// ---- MODULE/ACTOR_VALVE/PNEUMATIC_ACTOR/VISU/VisuCylinderHorLeft.TcVIS
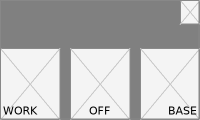
VISUALIZATION VisuCylinderHorLeft  // 200x120
VAR_IN_OUT
	fbVisuCylinder: FB_VISU_CYLINDER;
END_VAR
    Textfield (0,15 200x20), "%s", text variable: fbVisuCylinder.strInfo, colour toggle: fbVisuCylinder.stEvent.bEventActive
    Textfield (0,0 200x14), "%s", text variable: fbVisuCylinder.strFullObjName
    Image (143,85 52x30), invisible if: fbVisuCylinder.bBaseArrowInvisible, image: VisuSymbols.Symbols.ArrowBoldRight
        p2175578022: fbVisuCylinder.dwFrameColorBase
    Image (85,85 52x30), invisible if: fbVisuCylinder.bWorkArrowInvisible, image: VisuSymbols.Symbols.ArrowBoldLeft
        p2175578022: fbVisuCylinder.dwFrameColorWork
    Group (90,35 105x40)
        p3560616238: fbVisuCylinder.iMove
        RoundedRectangle (-10,10 100x20)
        RoundedRectangle (80,0 20x40)
    Rectangle (85,35 105x40)
        OnMouseClick: execute { fbVisuCylinder.bFrameInvisible:=false; }
    Frame (0,0 200x120), invisible if: fbVisuCylinder.bFrameInvisible, frame switch variable: fbVisuCylinder.iFrame
        shows VisuCylinderHorLeftCtrl(fbVisuCylinder := fbVisuCylinder)
END_VISUALIZATION

// ---- MODULE/ACTOR_VALVE/PNEUMATIC_ACTOR/VISU/VisuCylinderHorLeftCtrl.TcVIS
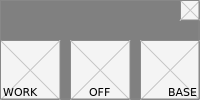
VISUALIZATION VisuCylinderHorLeftCtrl  // 200x100
VAR_IN_OUT
	fbVisuCylinder: FB_VISU_CYLINDER;
END_VAR
    Rectangle (0,0 200x100)
    Image (140,40 60x60), "BASE", image: VisuSymbols.Symbols.TriangleRight
        OnMouseClick: execute {
            fbVisuCylinder.bMoveToBase:=TRUE;
            fbVisuCylinder.bMoveToWork:=FALSE;
            fbVisuCylinder.bAllOff:=false;
            fbVisuCylinder.bFrameInvisible:= true;
        }
    Image (0,40 60x60), "WORK", image: VisuSymbols.Symbols.TriangleLeft
        OnMouseClick: execute {
            fbVisuCylinder.bMoveToWork:=TRUE;
            fbVisuCylinder.bMoveToBase:=FALSE;
            fbVisuCylinder.bAllOff:=false;
            fbVisuCylinder.bFrameInvisible:= true;
        }
    Image (180,0 20x20), image: VisuSymbols.Symbols.Wrong
        OnMouseDown: execute { fbVisuCylinder.bFrameInvisible:= true; }
    Image (70,40 60x60), "OFF", image: VisuSymbols.Symbols.Stop
        OnMouseClick: execute {
            fbVisuCylinder.bMoveToBase:=FALSE;
            fbVisuCylinder.bMoveToWork:=FALSE;
            fbVisuCylinder.bAllOff:=TRUE;
            fbVisuCylinder.bFrameInvisible:= true;
        }
END_VISUALIZATION

// ---- MODULE/ACTOR_VALVE/PNEUMATIC_ACTOR/VISU/VisuCylinderHorRight.TcVIS
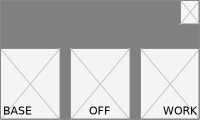
VISUALIZATION VisuCylinderHorRight  // 200x120
VAR_IN_OUT
	fbVisuCylinder: FB_VISU_CYLINDER;
END_VAR
    Textfield (0,15 200x20), "%s", text variable: fbVisuCylinder.strInfo, colour toggle: fbVisuCylinder.stEvent.bEventActive
    Textfield (0,0 200x14), "%s", text variable: fbVisuCylinder.strFullObjName
    Image (60,80 50x30), invisible if: fbVisuCylinder.bWorkArrowInvisible, image: VisuSymbols.Symbols.ArrowBoldRight
        p2175578022: fbVisuCylinder.dwFrameColorWork
    Image (5,80 50x30), invisible if: fbVisuCylinder.bBaseArrowInvisible, image: VisuSymbols.Symbols.ArrowBoldLeft
        p2175578022: fbVisuCylinder.dwFrameColorBase
    Group (5,30 100x40)
        p3560616238: fbVisuCylinder.iNegMove
        RoundedRectangle (0,10 100x20)
        RoundedRectangle (0,0 20x40)
    Rectangle (0,30 100x40)
        OnMouseClick: execute { fbVisuCylinder.bFrameInvisible:=false; }
    Frame (0,0 200x120), invisible if: fbVisuCylinder.bFrameInvisible, frame switch variable: fbVisuCylinder.iFrame
        shows VisuCylinderHorRightCtrl(fbVisuCylinder := fbVisuCylinder)
END_VISUALIZATION

// ---- MODULE/ACTOR_VALVE/PNEUMATIC_ACTOR/VISU/VisuCylinderHorRightCtrl.TcVIS
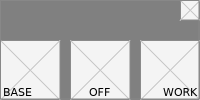
VISUALIZATION VisuCylinderHorRightCtrl  // 200x100
VAR_IN_OUT
	fbVisuCylinder: FB_VISU_CYLINDER;
END_VAR
    Rectangle (0,0 200x100)
    Image (140,40 60x60), "WORK", image: VisuSymbols.Symbols.TriangleRight
        OnMouseClick: execute {
            fbVisuCylinder.bMoveToBase:=FALSE;
            fbVisuCylinder.bMoveToWork:=true;
            fbVisuCylinder.bAllOff:=false;
            fbVisuCylinder.bFrameInvisible:= true;
        }
    Image (0,40 60x60), "BASE", image: VisuSymbols.Symbols.TriangleLeft
        OnMouseClick: execute {
            fbVisuCylinder.bMoveToWork:=FALSE;
            fbVisuCylinder.bMoveToBase:=true;
            fbVisuCylinder.bAllOff:=false;
            fbVisuCylinder.bFrameInvisible:= true;
        }
    Image (180,0 20x20), image: VisuSymbols.Symbols.Wrong
        OnMouseDown: execute { fbVisuCylinder.bFrameInvisible:= true; }
    Image (70,40 60x60), "OFF", image: VisuSymbols.Symbols.Stop
        OnMouseClick: execute {
            fbVisuCylinder.bMoveToBase:=FALSE;
            fbVisuCylinder.bMoveToWork:=FALSE;
            fbVisuCylinder.bAllOff:=TRUE;
            fbVisuCylinder.bFrameInvisible:= true;
        }
END_VISUALIZATION

// ---- MODULE/ACTOR_VALVE/PNEUMATIC_ACTOR/VISU/VisuCylinderHorRight_MidPos.TcVIS
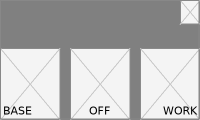
VISUALIZATION VisuCylinderHorRight_MidPos  // 200x120
VAR_IN_OUT
	fbVisuCylinder: FB_VISU_CYLINDER;
END_VAR
    Textfield (0,15 200x20), "%s", text variable: fbVisuCylinder.strInfo, colour toggle: fbVisuCylinder.stEvent.bEventActive
    Textfield (0,0 200x14), "%s", text variable: fbVisuCylinder.strFullObjName
    Image (75,80 30x30), invisible if: fbVisuCylinder.bWorkArrowInvisible, image: VisuSymbols.Symbols.ArrowBoldRight
        p2175578022: fbVisuCylinder.dwFrameColorWork
    Image (5,80 30x30), invisible if: fbVisuCylinder.bBaseArrowInvisible, image: VisuSymbols.Symbols.ArrowBoldLeft
        p2175578022: fbVisuCylinder.dwFrameColorBase
    Group (5,30 100x40)
        p3560616238: fbVisuCylinder.iNegMove
        RoundedRectangle (0,10 100x20)
        RoundedRectangle (0,0 20x40)
    Rectangle (0,30 100x40)
        OnMouseClick: execute { fbVisuCylinder.bFrameInvisible:=false; }
    Image (40,80 30x30), invisible if: fbVisuCylinder.bMidkArrowInvisible, image: VisuSymbols.Symbols.Bracket2
        p2175578022: fbVisuCylinder.dwFrameColorMid
    Frame (0,0 200x120), invisible if: fbVisuCylinder.bFrameInvisible, frame switch variable: fbVisuCylinder.iFrame
        shows VisuCylinderHorRightCtrl(fbVisuCylinder := fbVisuCylinder)
END_VISUALIZATION

// ---- MODULE/ACTOR_VALVE/PNEUMATIC_ACTOR/VISU/VisuCylinderTurn.TcVIS
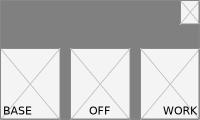
VISUALIZATION VisuCylinderTurn  // 200x120
VAR_IN_OUT
	fbVisuCylinder: FB_VISU_CYLINDER;
END_VAR
    Textfield (0,15 200x20), "%s", text variable: fbVisuCylinder.strInfo, colour toggle: fbVisuCylinder.stEvent.bEventActive
    Textfield (0,0 200x14), "%s", text variable: fbVisuCylinder.strFullObjName
    Image (145,65 50x50), invisible if: fbVisuCylinder.bWorkArrowInvisible, image: VisuSymbols.Symbols.ArrowHalfRightDown
        p2175578022: fbVisuCylinder.dwFrameColorWork
    Image (5,65 50x50), invisible if: fbVisuCylinder.bBaseArrowInvisible, image: VisuSymbols.Symbols.ArrowHalfLeftRight
        p2175578022: fbVisuCylinder.dwFrameColorBase
    RoundedRectangle (40,55 120x20)
        p2858320360: fbVisuCylinder.iAngle
    Ellipse (75,40 50x50)
        OnMouseClick: execute { fbVisuCylinder.bFrameInvisible:=false; }
    Frame (0,0 200x120), invisible if: fbVisuCylinder.bFrameInvisible, frame switch variable: fbVisuCylinder.iFrame
        shows VisuCylinderHorRightCtrl(fbVisuCylinder := fbVisuCylinder)
END_VISUALIZATION

// ---- MODULE/ACTOR_VALVE/PNEUMATIC_ACTOR/VISU/VisuCylinderVertDown.TcVIS
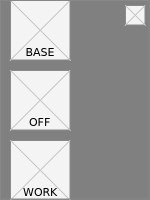
VISUALIZATION VisuCylinderVertDown  // 150x200
VAR_IN_OUT
	fbVisuCylinder: FB_VISU_CYLINDER;
END_VAR
    Image (85,85 30x50), invisible if: fbVisuCylinder.bWorkArrowInvisible, image: VisuSymbols.Symbols.ArrowBoldDown
        p2175578022: fbVisuCylinder.dwFrameColorWork
    Image (85,30 30x50), invisible if: fbVisuCylinder.bBaseArrowInvisible, image: VisuSymbols.Symbols.ArrowBoldUp
        p2175578022: fbVisuCylinder.dwFrameColorBase
    Group (25,40 40x100)
        p2738717112: fbVisuCylinder.iNegMove
        RoundedRectangle (10,0 20x100)
        RoundedRectangle (0,0 40x20)
    Rectangle (25,35 40x100)
        OnMouseClick: execute { fbVisuCylinder.bFrameInvisible:=false; }
    Textfield (0,15 150x20), "%s", text variable: fbVisuCylinder.strInfo, colour toggle: fbVisuCylinder.stEvent.bEventActive
    Textfield (0,0 150x14), "%s", text variable: fbVisuCylinder.strFullObjName
    Frame (0,0 150x200), invisible if: fbVisuCylinder.bFrameInvisible, frame switch variable: fbVisuCylinder.iFrame
        shows VisuCylinderVertDownCtrl(fbVisuCylinder := fbVisuCylinder)
END_VISUALIZATION

// ---- MODULE/ACTOR_VALVE/PNEUMATIC_ACTOR/VISU/VisuCylinderVertDownCtrl.TcVIS
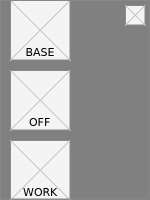
VISUALIZATION VisuCylinderVertDownCtrl  // 150x200
VAR_IN_OUT
	fbVisuCylinder: FB_VISU_CYLINDER;
END_VAR
    Rectangle (0,0 150x200)
    Image (10,140 60x60), "WORK", image: VisuSymbols.Symbols.TriangleDown
        OnMouseClick: execute {
            fbVisuCylinder.bMoveToBase:=FALSE;
            fbVisuCylinder.bMoveToWork:=true;
            fbVisuCylinder.bAllOff:=false;
            fbVisuCylinder.bFrameInvisible:= true;
        }
    Image (10,0 60x60), "BASE", image: VisuSymbols.Symbols.TriangleUp
        OnMouseClick: execute {
            fbVisuCylinder.bMoveToWork:=FALSE;
            fbVisuCylinder.bMoveToBase:=true;
            fbVisuCylinder.bAllOff:=false;
            fbVisuCylinder.bFrameInvisible:= true;
        }
    Image (125,5 20x20), image: VisuSymbols.Symbols.Wrong
        OnMouseDown: execute { fbVisuCylinder.bFrameInvisible:= true; }
    Image (10,70 60x60), "OFF", image: VisuSymbols.Symbols.Stop
        OnMouseClick: execute {
            fbVisuCylinder.bMoveToBase:=FALSE;
            fbVisuCylinder.bMoveToWork:=FALSE;
            fbVisuCylinder.bAllOff:=TRUE;
            fbVisuCylinder.bFrameInvisible:= true;
        }
END_VISUALIZATION

// ---- MODULE/ACTOR_VALVE/PNEUMATIC_ACTOR/VISU/VisuCylinderVertUp.TcVIS
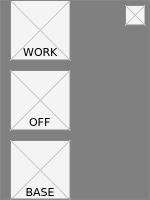
VISUALIZATION VisuCylinderVertUp  // 150x200
VAR_IN_OUT
	fbVisuCylinder: FB_VISU_CYLINDER;
END_VAR
    Image (85,90 30x50), invisible if: fbVisuCylinder.bWorkArrowInvisible, image: VisuSymbols.Symbols.ArrowBoldUp
        p2175578022: fbVisuCylinder.dwFrameColorWork
    Image (85,145 30x50), invisible if: fbVisuCylinder.bBaseArrowInvisible, image: VisuSymbols.Symbols.ArrowBoldDown
        p2175578022: fbVisuCylinder.dwFrameColorBase
    Group (25,90 40x100)
        p2738717112: fbVisuCylinder.iMove
        RoundedRectangle (10,0 20x100)
        RoundedRectangle (0,80 40x20)
    Rectangle (25,95 40x100)
        OnMouseClick: execute { fbVisuCylinder.bFrameInvisible:=false; }
    Textfield (0,15 150x20), "%s", text variable: fbVisuCylinder.strInfo, colour toggle: fbVisuCylinder.stEvent.bEventActive
    Textfield (0,0 150x14), "%s", text variable: fbVisuCylinder.strFullObjName
    Frame (0,0 150x200), invisible if: fbVisuCylinder.bFrameInvisible, frame switch variable: fbVisuCylinder.iFrame
        shows VisuCylinderVertUpCtrl(fbVisuCylinder := fbVisuCylinder)
END_VISUALIZATION

// ---- MODULE/ACTOR_VALVE/PNEUMATIC_ACTOR/VISU/VisuCylinderVertUpCtrl.TcVIS
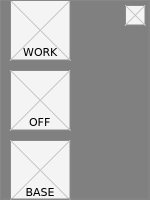
VISUALIZATION VisuCylinderVertUpCtrl  // 150x200
VAR_IN_OUT
	fbVisuCylinder: FB_VISU_CYLINDER;
END_VAR
    Rectangle (0,0 150x200)
    Image (10,0 60x60), "WORK", image: VisuSymbols.Symbols.TriangleUp
        OnMouseClick: execute {
            fbVisuCylinder.bMoveToBase:=FALSE;
            fbVisuCylinder.bMoveToWork:=true;
            fbVisuCylinder.bAllOff:=false;
            fbVisuCylinder.bFrameInvisible:= true;
        }
    Image (10,140 60x60), "BASE", image: VisuSymbols.Symbols.TriangleDown
        OnMouseClick: execute {
            fbVisuCylinder.bMoveToWork:=FALSE;
            fbVisuCylinder.bMoveToBase:=true;
            fbVisuCylinder.bAllOff:=false;
            fbVisuCylinder.bFrameInvisible:= true;
        }
    Image (125,5 20x20), image: VisuSymbols.Symbols.Wrong
        OnMouseDown: execute { fbVisuCylinder.bFrameInvisible:= true; }
    Image (10,70 60x60), "OFF", image: VisuSymbols.Symbols.Stop
        OnMouseClick: execute {
            fbVisuCylinder.bMoveToBase:=FALSE;
            fbVisuCylinder.bMoveToWork:=FALSE;
            fbVisuCylinder.bAllOff:=TRUE;
            fbVisuCylinder.bFrameInvisible:= true;
        }
END_VISUALIZATION

// ---- MODULE/BUS_DIAG/VISU/VISU_BUS_DIAG_MASTER.TcVIS
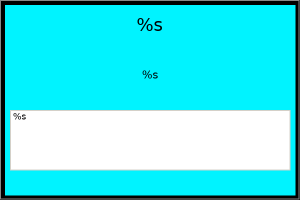
VISUALIZATION VISU_BUS_DIAG_MASTER  // 300x200
VAR_IN_OUT
	fbVisu: FB_VISU_BUS_DIAG;
END_VAR
    Rectangle (0,0 300x200), colour variable: fbVisu.dwColor
        p3450524324: fbVisu.dwColorFrame
    Textfield (10,10 280x30), "%s", text variable: fbVisu.strType
    Textfield (10,60 280x30), "%s", text variable: fbVisu.strName
    Textfield (10,110 280x60), "%s", text variable: fbVisu.strState
END_VISUALIZATION

// ---- MODULE/BYTES_TO_WORD/VISU/VISU_WORD_TO_BYTES.TcVIS
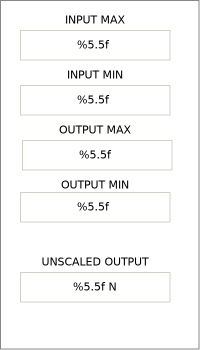
VISUALIZATION VISU_WORD_TO_BYTES  // 200x350
VAR_IN_OUT
	fbVISU:				FB_VISU_WORD_TO_BYTES;
END_VAR
    Textfield (20,30 150x30), "%5.5f", text variable: fbVISU.lrXMax
        OnMouseClick: write the text variable via Default, min 0, max 16085
    Label (20,5 150x30), "INPUT MAX"
    Textfield (20,85 150x30), "%5.5f", text variable: fbVISU.lrXMin
        OnMouseClick: write the text variable via Default, min 0, max 16085
    Label (20,60 150x30), "INPUT MIN"
    Textfield (22,140 150x30), "%5.5f", text variable: fbVISU.lrYMax
        OnMouseClick: write the text variable via Default, min 0
    Label (20,115 150x30), "OUTPUT MAX"
    Textfield (20,192 150x30), "%5.5f", text variable: fbVISU.lrYMin
        OnMouseClick: write the text variable via Default, min 0
    Label (20,170 150x30), "OUTPUT MIN"
    Textfield (20,272 150x30), "%5.5f N", text variable: fbVISU.lrUnscaledInput
        OnMouseClick: write the text variable via Default, min 0
    Label (20,247 150x30), "UNSCALED OUTPUT"
END_VISUALIZATION

// ---- ORGANISATION/OP_MODE/TXTLIST/TXT_LIST_OP_MODE.TcTLO
TEXTLIST TXT_LIST_OP_MODE
  7 = 'NOT-HALT' | en: 'EMERGANCY-STOP' | de: 'NOT-HALT' | zh_CHS: '急停'
  8 = 'MASCHINEN-FEHLER' | en: 'FATAL ERROR' | de: 'MASCHINEN-FEHLER' | zh_CHS: '致命错误'
  9 = 'STEUERUNG EIN' | en: 'CONTROL ON' | de: 'STEUERUNG EIN' | zh_CHS: '控制开启'
  1 = 'AUTOMATIK ' | en: 'AUTOMATIC' | de: 'AUTOMATIK ' | zh_CHS: '自动'
  2 = 'HANDBETRIEB' | en: 'MANUAL MODE' | de: 'HANDBETRIEB' | zh_CHS: '手动模式'
  3 = 'TIPPBETRIEB' | en: 'DEBUG MODE' | de: 'TIPPBETRIEB' | zh_CHS: 'DEBUG MODE'
  4 = 'GRUNDSTELLUNGSFAHRT' | en: 'INITIAL POS RIDE' | de: 'GRUNDSTELLUNGSFAHRT' | zh_CHS: '复位'
  5 = 'GRUNDSTELLUNG ERREICHT' | en: 'INITIAL POS REACH' | de: 'GRUNDSTELLUNG ERREICHT' | zh_CHS: '达成基本要求'
  101 = 'GST' | en: 'INIT' | de: 'GST' | zh_CHS: '的INIT'
  102 = 'AUTO' | en: 'AUTO' | de: 'AUTO' | zh_CHS: '自动'
  103 = 'HAND' | en: 'MANUAL' | de: 'HAND' | zh_CHS: '手册'
  104 = 'TIPP' | en: 'DEBUG' | de: 'TIPP' | zh_CHS: '去调查'
  105 = 'START' | en: 'START' | de: 'START' | zh_CHS: '开始'
  106 = 'STOP' | en: 'STOP' | de: 'STOP' | zh_CHS: '停'
  11 = 'VORWAHL AUTOMATIK' | en: 'SELECTION AUTOMATIC' | de: 'VORWAHL AUTOMATIK' | zh_CHS: '自动选择'
  12 = 'VORWAHL HAND' | en: 'SELECTION MANUAL' | de: 'VORWAHL HAND' | zh_CHS: '选择手册'
  13 = 'VORWAHL TIPPBETRIEB' | en: 'SELECTION DEBUG' | de: 'VORWAHL TIPPBETRIEB' | zh_CHS: '选择调试'
  14 = 'VORWAHL GRUNDSTELLUNGSFAHRT' | en: 'SLECTION INITIAL POS RIDE' | de: 'VORWAHL GRUNDSTELLUNGSFAHRT' | zh_CHS: '选择初始POS RIDE'
  0 = 'MASCHINE EINSCHALTEN' | en: 'TURN ON THE MACHINE' | de: 'MASCHINE EINSCHALTEN' | zh_CHS: '启动机器'
  107 = 'PAUSE' | en: 'PAUSE' | de: 'PAUSE'
  6 = 'PAUSE' | en: 'PAUSE' | de: 'PAUSE'
  10 = 'DRUCK OK' | en: 'DRUCK OK' | de: 'MAIN AIR OK'
   = ''
END_TEXTLIST

// ---- TXT_LIST_OBJECTS.TcTLO
TEXTLIST TXT_LIST_OBJECTS
  _3627.PLC_851.PrgStation.fbPowerAdapter1 = 'Netzteil 1' | de: 'Maschine' | en: 'Maschine'
  _3627.PLC_851.PrgStation.fbPowerAdapter2 = 'Netzteil 2' | de: 'Not-Halt links' | en: 'E-Stop left'
  _3627.PLC_851.PrgStation.fbZylinderLinks = 'Zylinder Links' | de: 'Not-Halt rechts' | en: 'E-Stop right'
  _3627.PLC_851.PrgStation.fbZylinderRechts = 'Zylinder Rechts' | de: 'Schutztür oben' | en: 'Door left'
  _3627.PLC_851.PrgStation.fbCalibrateVoltageInput1 = 'Scallieren Spannung (V)' | de: 'Schutztür rechts' | en: 'Door right'
  _3627.PLC_851.PrgStation.fbCalibrateVoltageInput2 = 'Scallieren Spannung (V)' | de: 'Maschine' | en: 'Machine'
  _3627.PLC_851.PrgStation.fbCalibrateCurrentInput1 = 'Scallieren Strom (A)' | de: 'Vakuum Druckstück' | en: 'Sensor 1'
  _3627.PLC_851.PrgStation.fbCalibrateCurrentInput2 = 'Scallieren Strom (A)' | de: 'Vakuum Druckpilz' | en: 'Vac Syst 1'
  _3531.PLC_851.PrgStation.fbStepSeqFindZeroPosPolepiece = 'Nullpunkt Suche Druckstück' | de: 'Nullpunkt-Suche Druckstück'
  _3531.PLC_851.PrgStation.fbStepSeqFindZeroPosPole = 'Nullpunkt Suche Stange' | de: 'Nullpunkt-Suche Stange'
  _3531.PLC_851.PrgStation.fbScanner = 'Scanner Druckstück' | de: 'Scanner Druckstück' | en: 'Scan Polepiece'
  _3531.PLC_851.PrgStation.fbECMaster = 'Beckoff PC' | de: 'Beckoff PC'
  _3531.PLC_851.PrgStation.fbPress = 'Kistler Presse' | de: 'Kistler Presse'
  _3531.PLC_851.PrgStation.fbCamera1 = 'Kamera Druckstange' | de: 'Kamera Druckstange' | en: 'Camera 1'
  _3531.PLC_851.PrgStation.fbCamera2 = 'Kamera Druckpilz' | de: 'Kamera Druckpilz' | en: 'Camera 2'
  _3531.PLC_851.PrgStation.fbGripper1 = 'Greifer links' | de: 'Greifer links'
  _3531.PLC_851.PrgStation.fbGripper2 = 'Greifer rechts' | de: 'Greifer rechts'
  _3531.PLC_851.PrgStation.fbAxisDruckstangeFunktions = 'Schrittmotor Druckstange' | de: 'Schrittmotor Druckstange'
  _3531.PLC_851.PrgStation.fbAxisDruckstueckFunctions = 'Schrittmotor Druckstück' | de: 'Schrittmotor Druckstück'
   = ''
END_TEXTLIST
